(* PLC project Unnamed, Unknown Unnamed 1 *)
(* stored: creationDateTime 2024-12-08T23:22:04, modificationDateTime 2024-12-16T12:34:26 *)

PROGRAM Main
  VAR
    AA1 : BOOL;
    AA2 : BOOL;
    AA3 : BOOL;
  END_VAR

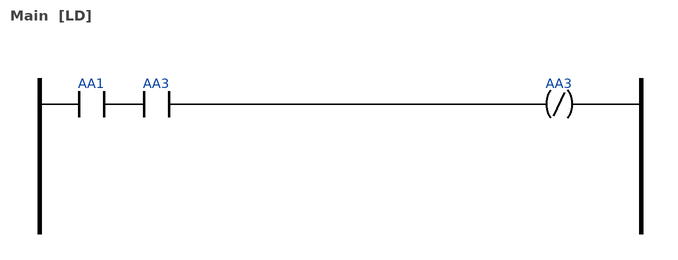
(* LD diagram, written out as Structured Text *)
AA3 := NOT (AA1 AND AA3);
END_PROGRAM

CONFIGURATION Config0
  RESOURCE Res0 ON PLC
    TASK task0(INTERVAL := T#20ms, PRIORITY := 0);
    PROGRAM instance0 WITH task0 : Main;
  END_RESOURCE
END_CONFIGURATION
